// TIA Portal V17 export
// export: Created 2024-09-03T21:54:51.865258Z, ExportSetting WithDefaults, DisplayName Totally Integrated Automation Portal, DisplayVersion V17 Update 7, DisplayName TIA Portal Openness, DisplayVersion V17 Update 7, DisplayName TIA Portal Version Control Interface, DisplayVersion V17, DisplayName SINAMICS Startdrive Advanced, DisplayVersion V17 SP2, DisplayName SINAMICS Startdrive G110M, G120, G120C, G120D, G120P, G115D, DisplayVersion V17 SP2, DisplayName SINAMICS Startdrive G130, G150, S120, S150, SINAMICS MV, S210, DisplayVersion V17 SP2, DisplayName STEP 7 Professional, DisplayVersion V17 Update 7, DisplayName STEP 7 Safety, DisplayVersion V17 Update 6, DisplayName WinCC Advanced / Unified PC, DisplayVersion V17 Update 7
FUNCTION_BLOCK "Readings"   // FB300, LAD
{ S7_Optimized_Access := 'TRUE' }
VERSION : 0.1
// stored: AutoNumber false, IsIECCheckEnabled false, IsRetainMemResEnabled false, MemoryReserve 100, SetENOAutomatically false, UDAEnableTagReadback false
   VAR
      Stat : Struct
         Init : Bool;
         Run : Bool;
         Process : Bool;
      END_STRUCT;
   END_VAR
   VAR_TEMP
      i : Int;
   END_VAR
BEGIN

REGION Network 2 (SCL)
   FOR #i := 1 TO "MaxReader" DO
       IF "DB_ProductionProgramActual".Program.Readings[#i].Enable THEN
           IF "DB_ProductionProgramActual".Program.Readings[#i].ReaderNumber > 0 THEN
               "Reader Cognex Dataman"("Reader Parameters".Reader["DB_ProductionProgramActual".Program.Readings[#i].ReaderNumber]);



               ;
           END_IF;


       END_IF;

       ;
   END_FOR;
END_REGION
END_FUNCTION_BLOCK
